TYPE ST_Netze_Parameter :
STRUCT
	Kaltwasser		: ST_ThNTZ_Parameter;
	Warmwasser		: ST_ThNTZ_Parameter;
	Heisswasser		: ST_ThNTZ_Parameter;
END_STRUCT
END_TYPE

(* stored: Version 1.1.0.1, ProductVersion 3.1.4024.9
   DUT ST_Netze_Parameter: Id {dda06e2c-5077-4e72-825f-d2d643b6bea0} *)
